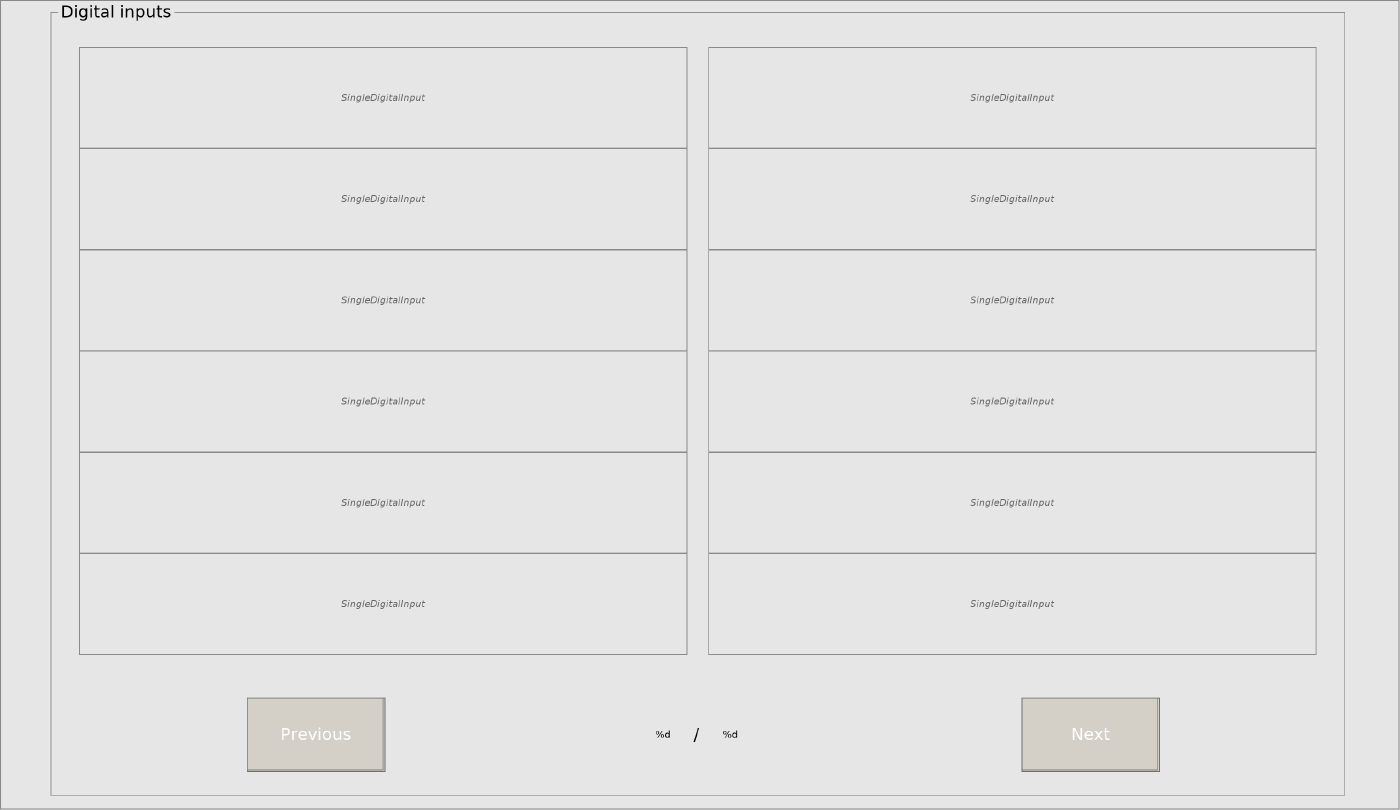
VISUALIZATION PageManualInputs_1  // 1520x880
VAR_IN_OUT
	btnPrevious			: BOOL;
	btnNext				: BOOL;
	
	bPreviousInvisible	: BOOL;
	bNextInvisible		: BOOL;
	
	stDigitalInputEmpty	: ARRAY[1..12] OF BOOL;
	stDigitalInputData	: ARRAY[1..12] OF ST_VisuCtrlInputFrame;
	
	iInputSelectedPageIndex		: USINT;
	iInputTotalPageIndex 		: USINT;
END_VAR
    GroupBox (55,5 1405x859), "Digital inputs"
        Rectangle (713,768 50x50), "%d", text variable: iInputTotalPageIndex+1
        Rectangle (640,768 50x50), "%d", text variable: iInputSelectedPageIndex+1
        Rectangle (636,768 130x50), "/"
        Button (213,753 150x80), "Previous", invisible if: bPreviousInvisible
            tap btnPrevious
        Button (1054,753 150x80), "Next", invisible if: bNextInvisible
            tap btnNext
        Frame (31,46 660x110), invisible if: stDigitalInputEmpty[1]
            shows SingleDigitalInput(stDigitalInput := stDigitalInputData[1])
        Frame (31,156 660x110), invisible if: stDigitalInputEmpty[2]
            shows SingleDigitalInput(stDigitalInput := stDigitalInputData[2])
        Frame (31,266 660x110), invisible if: stDigitalInputEmpty[3]
            shows SingleDigitalInput(stDigitalInput := stDigitalInputData[3])
        Frame (31,376 660x110), invisible if: stDigitalInputEmpty[4]
            shows SingleDigitalInput(stDigitalInput := stDigitalInputData[4])
        Frame (31,486 660x110), invisible if: stDigitalInputEmpty[5]
            shows SingleDigitalInput(stDigitalInput := stDigitalInputData[5])
        Frame (31,596 660x110), invisible if: stDigitalInputEmpty[6]
            shows SingleDigitalInput(stDigitalInput := stDigitalInputData[6])
        Frame (714,46 660x110), invisible if: stDigitalInputEmpty[7]
            shows SingleDigitalInput(stDigitalInput := stDigitalInputData[7])
    Frame (769,161 660x110), invisible if: stDigitalInputEmpty[8]
        shows SingleDigitalInput(stDigitalInput := stDigitalInputData[8])
    Frame (769,271 660x110), invisible if: stDigitalInputEmpty[9]
        shows SingleDigitalInput(stDigitalInput := stDigitalInputData[9])
    Frame (769,381 660x110), invisible if: stDigitalInputEmpty[10]
        shows SingleDigitalInput(stDigitalInput := stDigitalInputData[10])
    Frame (769,491 660x110), invisible if: stDigitalInputEmpty[11]
        shows SingleDigitalInput(stDigitalInput := stDigitalInputData[11])
    Frame (769,601 660x110), invisible if: stDigitalInputEmpty[12]
        shows SingleDigitalInput(stDigitalInput := stDigitalInputData[12])
END_VISUALIZATION

(* stored: Version 1.1.0.1, ProductVersion 3.1.4024.12
   Visu PageManualInputs_1: Id {2fc2c7a4-c6b4-4ff0-94a5-1fb0b9fde0e9} *)
